TYPE ST_EBUS_AnalogueDataIn :
STRUCT
	nStatus		: WORD;
	nValue		: INT;
END_STRUCT
END_TYPE

(* stored: Version 1.1.0.1, ProductVersion 3.1.4024.15
   DUT ST_EBUS_AnalogueDataIn: Id {ace872fc-a4e9-4faf-a740-6e962ce85199} *)
